// TIA Portal V16 export
// export: Created 2022-01-12T14:32:04.3791802Z, ExportSetting WithDefaults, DisplayName Totally Integrated Automation Portal, DisplayVersion V16 Update 4, DisplayName TIA Portal Version Control Interface, DisplayVersion V16 Update 2, DisplayName TIA Portal Openness, DisplayVersion V16 Update 4, DisplayName STEP 7 Professional, DisplayVersion V16 Update 4, DisplayName STEP 7 Safety, DisplayVersion V16, DisplayName WinCC Professional, DisplayVersion V16 Update 4
DATA_BLOCK "DB_reports_mlekomat"   // DB12
{ S7_Optimized_Access := 'TRUE' }
VERSION : 0.1
// stored: AutoNumber true, DBAccessibleFromOPCUA true, IsOnlyStoredInLoadMemory false, IsRetainMemResEnabled false, IsWriteProtectedInAS false, MemoryReserve 100
   VAR RETAIN
      cips : Array[0..7] of Struct
         cip_active : Bool;   // teraz trwa mycie
         print_report : Bool;   // bit dla scady żeby wydrukowała raport
         print_report_done : Bool;   // bit ze skady ze raport się wydrukował
         number_of_cip : Int;   // aktualny numer kolejnego mycia w historii
         start_cip_date_and_time : Date_And_Time;
         start_lye_date_and_time : Date_And_Time;
         start_acid_date_and_time : Date_And_Time;
         start_disinfection_date_and_time : Date_And_Time;
         stop_cip_date_and_time : Date_And_Time;
      END_STRUCT;
   END_VAR
BEGIN
END_DATA_BLOCK
